Fanuc KAREL source: PATH_LEN.kl

PROGRAM T
%NOLOCKGROUP
VAR
 v0 : PATH
 res : INTEGER
BEGIN
 res = PATH_LEN(v0)
END T
